// Mitsubishi GX Works2 project: 알람   PLC: Q02/Q02H

PROGRAM MAIN
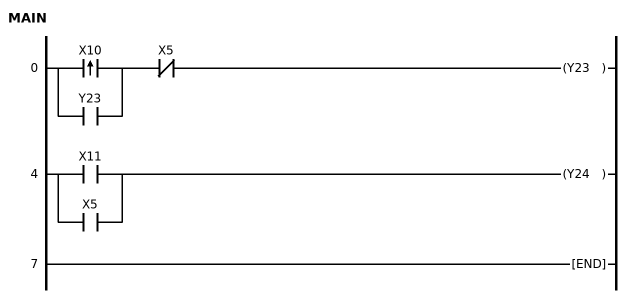
0     LDP     X10
      OR      Y23
      ANI     X5
      OUT     Y23
4     LD      X11
      OR      X5
      OUT     Y24
7     END
END_PROGRAM

PROGRAM HMI
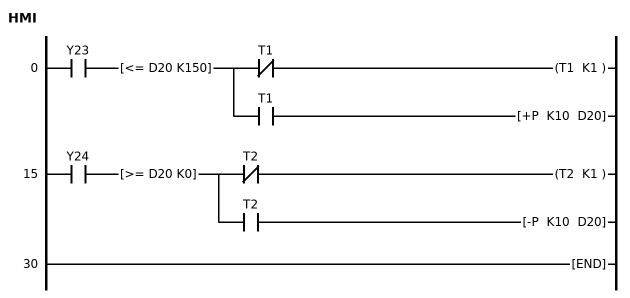
0     LD      Y23
      AND<=   D20 K150
      MPS
      ANI     T1
      OUT     T1 K1
      MPP
      AND     T1
      +P      K10 D20
15    LD      Y24
      AND>=   D20 K0
      MPS
      ANI     T2
      OUT     T2 K1
      MPP
      AND     T2
      -P      K10 D20
30    END
END_PROGRAM

PROGRAM HMI1
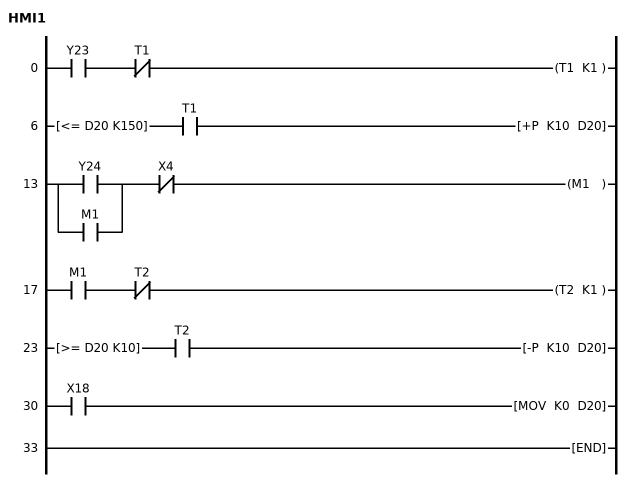
0     LD      Y23
      ANI     T1
      OUT     T1 K1
6     LD<=    D20 K150
      AND     T1
      +P      K10 D20
13    LD      Y24
      OR      M1
      ANI     X4
      OUT     M1
17    LD      M1
      ANI     T2
      OUT     T2 K1
23    LD>=    D20 K10
      AND     T2
      -P      K10 D20
30    LD      X18
      MOV     K0 D20
33    END
END_PROGRAM

PROGRAM ERR
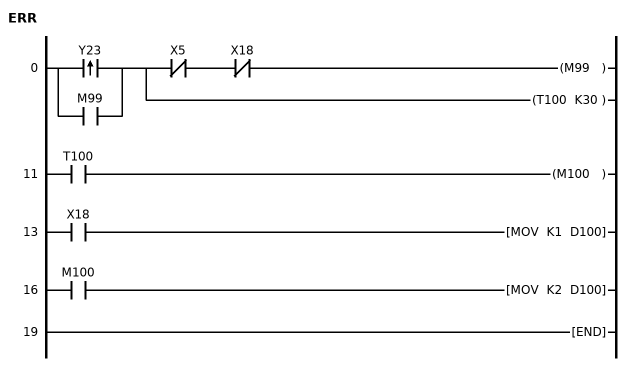
0     LDP     Y23
      OR      M99
      MPS
      ANI     X5
      ANI     X18
      OUT     M99
      MPP
      OUT     T100 K30
11    LD      T100
      OUT     M100
13    LD      X18
      MOV     K1 D100
16    LD      M100
      MOV     K2 D100
19    END
END_PROGRAM
